{attribute 'qualified_only'}
{attribute 'strict'}
TYPE CircuitBreakerStatus :
(
	OFF := 0,        // Device has been set OFF either manually or programatically
	ON := 1,		 // Device is ON and funcioning normally
	TRIPPED := 2,	 // An overcurrent event has tripped the device
	RESET := 3		 // A reset signal has been sent to the device but it hasn't responded yet
);
END_TYPE

(* stored: Version 1.1.0.1, ProductVersion 3.1.4024.15
   EnumerationTextList CircuitBreakerStatus: Id {dcbef35d-17b3-4961-88ee-70174408f427} *)
